{attribute 'qualified_only'}
{attribute 'strict'}
TYPE Trigger_Error :
(
	None := 0,
	Camera_Busy := 1,
	Camera_Not_Trigger_Redy := 2
) UINT;
END_TYPE

(* stored: Version 1.1.0.1, ProductVersion 3.1.4024.10
   DUT Trigger_Error: Id {8f72347c-78d0-4a33-b700-adf13de20256} *)
